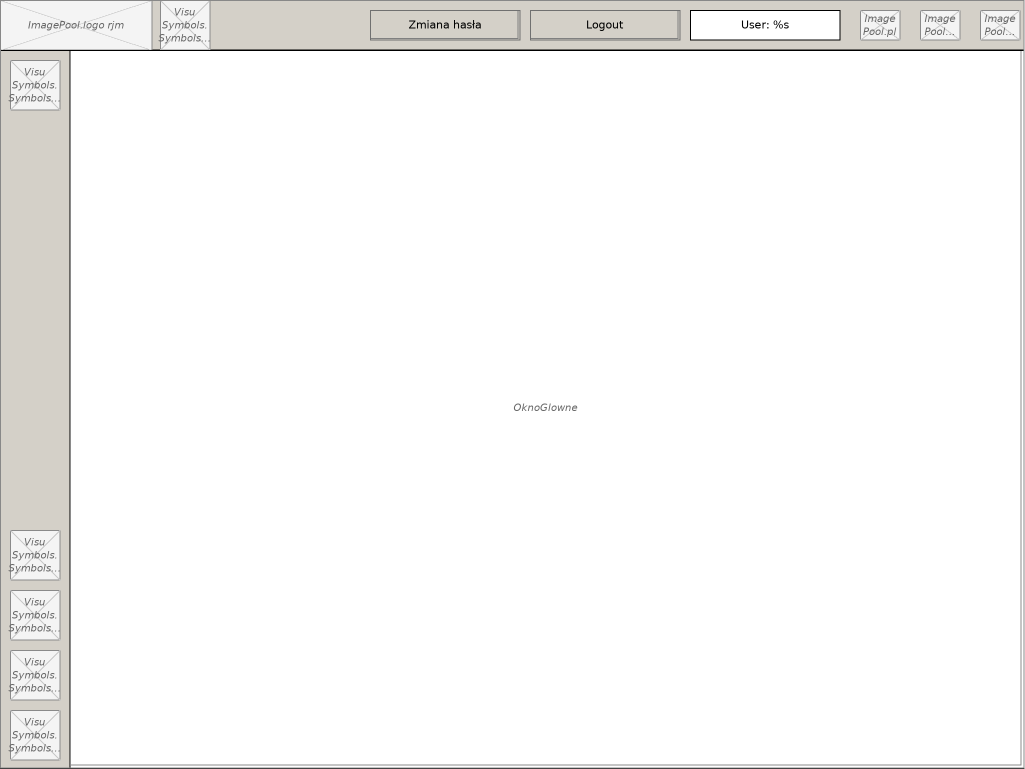
VISUALIZATION Visualization  // 1025x769
    Rectangle (0,0 1024x50)
    Rectangle (0,50 70x718)
    Frame (70,50 951x715), frame switch variable: GVL_Wizualizacja.iNumerRamki
        shows OknoGlowne()
        shows Visu_StanMaszyny_DiagramZPrzyciskami(bWlaczPrzyciski := GVL_StanMaszyny.bWlaczPrzyciski)
        shows Visu_LogowanieBledow_Tabela(stParametry := GVL_LogowanieBledow.fbLoger.stWyswietlanieParametry)
        shows Ustawienia()
    Button (10,60 50x50), colour toggle: GVL_Wizualizacja.iNumerRamki = 0
    Button (10,710 50x50), colour toggle: GVL_Wizualizacja.iNumerRamki = 2
    Button (10,650 50x50), colour toggle: GVL_Wizualizacja.iNumerRamki = 1
    Image (10,60 50x50), colour toggle: GVL_Wizualizacja.iNumerRamki = 0, image: VisuSymbols.Symbols.Home
        OnMouseDown: execute {
            GVL_Wizualizacja.iNumerRamki := 0;
            GVL_StanMaszyny.bWlaczPrzyciski := FALSE;
            GVL_LogowanieBledow.bWyswietlAlarmy := FALSE;
        }
    Image (10,650 50x50), image: VisuSymbols.Symbols.Information
        OnMouseDown: execute {
            GVL_Wizualizacja.iNumerRamki := 1;
            GVL_StanMaszyny.bWlaczPrzyciski := TRUE;
            GVL_LogowanieBledow.bWyswietlAlarmy := FALSE;
        }
    Image (10,710 50x50), image: VisuSymbols.Symbols.Security
        OnMouseDown: execute {
            GVL_Wizualizacja.iNumerRamki := 2;
            GVL_StanMaszyny.bWlaczPrzyciski := FALSE;
            GVL_LogowanieBledow.bWyswietlAlarmy := TRUE;
        }
    Image (160,0 50x50), image: VisuSymbols.Symbols.voltage
    Line (0,768) (1024,768)
    Line (1024,768) (1024,0)
    Button (10,590 50x50), colour toggle: GVL_Wizualizacja.iNumerRamki = 3
    Image (10,590 50x50), image: VisuSymbols.Symbols.ControlPanel
        OnMouseDown: execute {
            GVL_Wizualizacja.iNumerRamki := 3;
            GVL_StanMaszyny.bWlaczPrzyciski := FALSE;
            GVL_LogowanieBledow.bWyswietlAlarmy := FALSE;
        }
    Image (0,0 152x50), image: ImagePool.logo rjm
    Line (0,50) (1024,50)
    Image (920,10 40x30), image: ImagePool.de
        OnMouseDown: ChangeLanguage ChangeLanguage=DE
        OnMouseDown: execute { GVL_LogowanieBledow.fbLoger.iJezykID := 1031; }
    Image (980,10 40x30), image: ImagePool.gb
        OnMouseDown: ChangeLanguage ChangeLanguage=EN
        OnMouseDown: execute { GVL_LogowanieBledow.fbLoger.iJezykID := 1033; }
    Image (860,10 40x30), image: ImagePool.pl
        OnMouseDown: execute { GVL_LogowanieBledow.fbLoger.iJezykID := 1045; }
        OnMouseDown: ChangeLanguage ChangeLanguage=PL
    Button (530,10 150x30), "Login", invisible if: VisuElemsWinControls.CurrentUserName <> ""
        OnMouseDown: VisuUserMgmt Type=Login
    Button (530,10 150x30), "Logout", invisible if: VisuElemsWinControls.CurrentUserName = ""
        OnMouseDown: VisuUserMgmt Type=Logout
    Rectangle (690,10 150x30), "User: %s", text variable: VisuElemsWinControls.CurrentUserName
    Button (370,10 150x30), "Zmiana hasła"
        OnMouseDown: VisuUserMgmt Type=ChangeUserPassword
    Button (10,530 50x50)
    Image (10,530 50x50), image: VisuSymbols.Symbols.EditUser
        OnMouseDown: VisuUserMgmt Type=OpenUserConfiguration
END_VISUALIZATION

(* stored: Version 1.1.0.1, ProductVersion 3.1.4024.11
   Visu Visualization: Id {28aa2546-4191-4993-9a41-98daafec61d7} *)
